Fanuc KAREL source: kt00585.KL

PROGRAM KT00585
%STACKSIZE=65535
%PRIORITY=65535
%NOLOCKGROUP
VAR
I1 : INTEGER
-- UNRESOLVED DECLARATIONS (source type spelling not recovered)
-- V2 : TYPE_0x0013 (type_u16=0x0013)
-- OUT : TYPE_0x0013 (type_u16=0x0013)
BEGIN
I1=2
-- UNSAFE_SOURCE_IR line 9: field_offset(V2,4) = 1073741824
-- UNRESOLVED_PC line 10 opcodes [21 49 8B 4A] marker_code=36
END KT00585
